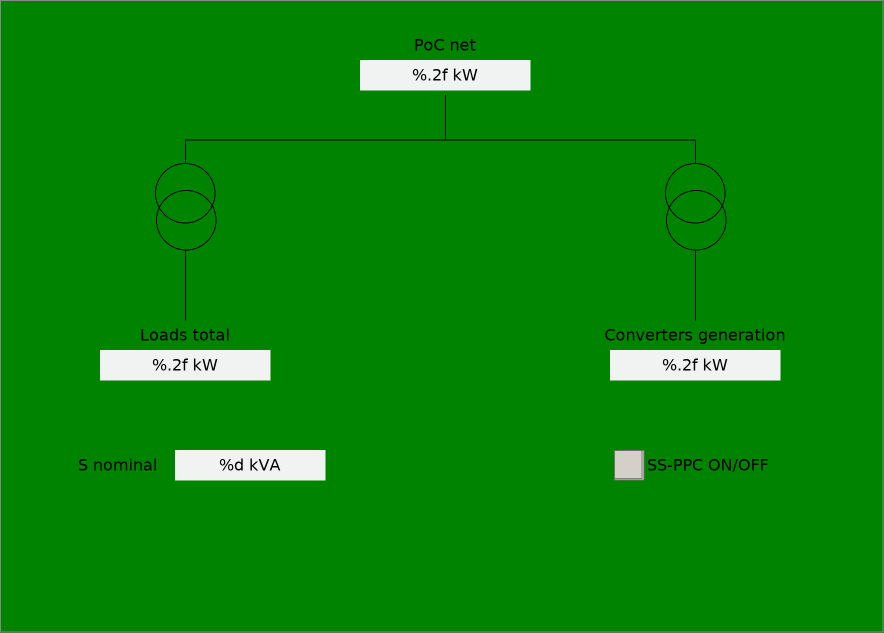
VISUALIZATION Main  // 884x633
    Rectangle (360,60 170x30), "%.2f kW", text variable: GVL_POWERMETER.M_board_P_kW
    Rectangle (390,30 110x30), "PoC net"
    Rectangle (610,350 170x30), "%.2f kW", text variable: GVL_POWERMETER.P_converters_tot
    Rectangle (605,320 180x30), "Converters generation"
    Rectangle (100,350 170x30), "%.2f kW", text variable: GVL_POWERMETER.M_board_P_kW + GVL_POWERMETER.P_converters_tot
    Rectangle (130,320 110x30), "Loads total"
    Line (445,95) (445,140)
    Line (695,250) (695,320)
    Line (185,250) (185,320)
    Ellipse (156,190 60x60)
    Ellipse (155,163 60x60)
    Ellipse (666,190 60x60)
    Ellipse (665,163 60x60)
    Line (695,140) (695,163)
    Line (185,140) (185,163)
    Line (695,140) (185,140)
    Rectangle (175,450 150x30), "%d kVA", text variable: GVL_PLANT_DEF.Plant_capacity_nom
        OnMouseClick: write the text variable via Default
    Rectangle (75,450 92x30), "S nominal"
    Rectangle (644,450 211x30), "SS-PPC ON/OFF"
    Button (614,450 30x30), colour toggle: GVL_GUI.Conv_n_mode_button[13]
        OnMouseClick: toggle GVL_GUI.Conv_n_mode_button[13]
        OnMouseClick: execute {
            IF GVL_CONV_COMMS.Night_Mode_Active[13] = 0 THEN
            	GVL_CONV_COMMS.Comms_Control_Word[13]:= GVL_CONV_COMMS.Comms_Control_Word[13] OR 16#0002;
            ELSE
            	GVL_CONV_COMMS.Comms_Control_Word[13]:= GVL_CONV_COMMS.Comms_Control_Word[13] AND 16#FFFD;
            END_IF
        }
END_VISUALIZATION

(* stored: Version 1.1.0.1, ProductVersion 3.1.4024.11
   Visu Main: Id {951b4d45-733f-4208-a5f2-b9bc82e80eab} *)
